(* CODESYS project LogData.gvl.xml

Project tree, tasks and I/O mapping:
  global variables LogData
*)

// LogData
{attribute 'qualified_only'}
VAR_GLOBAL
	Door: DoorLogData;
	Heater: HeaterLogData;
	Hopper: HopperLogData;
	IceMaker: IceMakerLogData;
END_VAR
